# EPICS autosave request: iocBoot/iocUSBTEMP-AI/auto_settings.req
file "USB_TEMP_settings.req", P=USB_TEMP:
